# EPICS substitutions: epics/db/EL9410.substitutions
file "./db/ecSlave.template"
{
  pattern {}
          {}
}

file "./db/EL9410.template"
{
  pattern {}
          {}
}
